// TIA Portal V20 export
TYPE "BarCode"
// stored: Access Published, Namespace Global
   STRUCT
      "Result Data" : Array[0..63] of Byte;
   END_STRUCT;
END_TYPE
